// note: 7 stored wires end on pins the file does not list and are not shown
BCV_Loop.DeadBand := SEL(BCV_Loop.DeadBand = 0.0, BCV_Loop.DeadBand, 0.1);
BCV_Loop.Live_Target_EU := SEL(BCV_Loop.Mode=Temp_Loop_Modes.Step, BCV_Loop.Target_EU, SEL(HEATING, TT.EU-(BCV_Loop.DeadBand*1.5), TT.EU+(BCV_Loop.DeadBand*1.5)));
_w1 := (BCV_Loop.Mode = Temp_Loop_Modes.Crash) OR (BCV_Loop.Mode = Temp_Loop_Modes.Step);
_w2 := ABS(BCV_Loop.Target_EU - TT.EU);
ABS_Error := _w2;
(* _w2 * BCV_Loop.kp < 50; result not used *)
TON_2(IN := False OR _w2 < BCV_Loop.Window, PT := T#5s); // TON
_w3 := _w1 AND TON_2.Q;
In_Zone := _w3;
R_TRIG_0(CLK := _w1 AND _w3); // R_trig
IF R_TRIG_0.Q THEN _w4 := Temp_Loop_Modes.Auto; END_IF
BCV_Loop.Mode := _w4;
_w5 := REAL_TO_TIME(BCV_LOOP.Min_Cycle_S) * 1000;
_w6 := On_Seconds > BCV_LOOP.Min_Cycle_S;
_w7 := SEL(Heating, BCV_Loop.Live_Target_EU, BCV_Loop.Actual_EU);
_w8 := SEL(Heating, BCV_Loop.Actual_EU, BCV_Loop.Live_Target_EU);
TOF_0(IN := Permisive, PT := T#15s); // TOF
TON_3(IN := TOF_0.Q, PT := T#15s); // TON
_w9 := On_Seconds > BCV_LOOP.Max_Cycle_S - BCV_LOOP.Min_Cycle_S;
SR_0(SET1 := Loop_Disable, RESET := BCV_Loop.Mode=Temp_Loop_Modes.Idle); // SR
TP_1(IN := _w3, PT := T#5s); // TP
IF SR_0.Q1 THEN _w10 := Temp_Loop_Modes.Idle; END_IF
BCV_Loop.Mode := _w10;
_w11 := UINT_TO_TIME(BCV_Loop.Timer_Target_M) * 60000;
TOF_1(IN := (TT.Status.eStatus=eSensor_Status.Offline) OR (TT.Status.eStatus=eSensor_Status.Fault), PT := t#15s); // TOF
_w12 := (BCV_Loop.Mode=Temp_Loop_Modes.Auto_Paused) OR (BCV_Loop.Mode=Temp_Loop_Modes.Idle) OR NOT TON_3.Q OR SR_0.Q1 OR (BCV_Loop.Status=Temp_Loop_Status.Timer_Expired) OR TOF_1.Q;
_w13 := _w12 OR (_w12 OR TP_1.Q);
PID_Reset := _w13;
FT_PIDW_0(
    IN := SEL(_w12, _w8, _w7) - _w7,
    KP := BCV_Loop.kp,
    TN := BCV_Loop.TN,
    TV := BCV_Loop.TV,
    LIM_L := 0,
    LIM_H := 100,
    RST := _w13); // BURKERT_OSCAT_BASIC.FT_PIDW
BCV_Loop.Limiter := FT_PIDW_0.LIM;
_w14 := SEL(PID_Reset, SEL(BCV_Loop.Mode=Temp_Loop_Modes.Crash, FT_PIDW_0.Y, 100.0), 0.0);
BCV_Loop.Load_EU := _w14;
_w15 := _w14 * ((BCV_Loop.Max_Cycle_S/100.0));
On_Seconds := _w15;
GEN_PULSE_0(
    ENQ := _w6,
    PTH := REAL_TO_TIME(_w15) * 1000,
    PTL := REAL_TO_TIME(BCV_LOOP.Max_Cycle_S - _w15) * 1000); // BURKERT_OSCAT_BASIC.GEN_PULSE
_w16 := _w6 AND GEN_PULSE_0.Q;
TP_0(IN := _w16, PT := _w5); // TP
_w17 := (TP_0.Q OR _w16 OR _w9) AND NOT Loop_Disable AND NOT (BCV_Loop.Mode=Temp_Loop_Modes.Idle);
BCV_Loop.Output := _w17;
BCV.PLC_CMD := _w17;
_w18 := (BCV_Loop.Mode=Temp_Loop_Modes.Profile) AND (BCV_Loop.Timer_Target_M>0) AND NOT _w13 AND NOT Profile_Reset;
TON_0(IN := _w18, PT := _w11); // TON
Current_Minute := TIME_TO_UINT(TON_0.ET / 60000);
BCV_Loop.Timer_Remaining_s := TIME_TO_UINT((_w11 - TON_0.ET) / 1000);
TT.Alarm_Config.Setpoints.Hi_Hi_Alarm := SEL(NOT _w12, TT.Alarm_Config.Setpoints.Hi_Hi_Alarm, BCV_Loop.Live_Target_EU+(BCV_Loop.Window*2));
_w19 := (TT.Status.eStatus=eSensor_Status.Offline) OR (TT.Status.eStatus=eSensor_Status.Offline);
Loop_Disable := External_Fault OR (TT.Status.eStatus=eSensor_Status.FORCED) OR (BCV.Mode<>eBCV_Modes.Auto) OR _w19;
TT.Alarm_Config.Setpoints.Hi_Warn := SEL(NOT _w12, TT.Alarm_Config.Setpoints.Hi_Warn, BCV_Loop.Live_Target_EU+(BCV_Loop.Window));
TT.Alarm_Config.Setpoints.Low_warn := SEL(NOT _w12, TT.Alarm_Config.Setpoints.Low_warn, BCV_Loop.Live_Target_EU-(BCV_Loop.Window));
TT.Alarm_Config.Setpoints.Low_Low_Alarm := SEL(NOT _w12, TT.Alarm_Config.Setpoints.Low_Low_Alarm, BCV_Loop.Live_Target_EU-(BCV_Loop.Window*2));
BCV_Loop.Status := SEL(BCV.Mode<>eBCV_Modes.Auto, SEL(TT.Status.eStatus=eSensor_Status.FORCED, SEL(External_Fault, SEL(_w19, SEL(BCV_Loop.Mode=Temp_Loop_Modes.Auto_Paused, SEL(BCV_Loop.Mode=Temp_Loop_Modes.Idle, SEL(TT.Status.eStatus=eSensor_Status.Low_Low_Alarm, SEL(TT.Status.eStatus=eSensor_Status.Low_Warning, SEL(TT.Status.eStatus=eSensor_Status.HiHi_Alarm, SEL(TT.Status.eStatus=eSensor_Status.High_Warning, SEL(TON_0.Q, SEL(_w18, SEL(BCV_Loop.Mode=Temp_Loop_Modes.Auto, SEL(Permisive, Temp_Loop_Status.Pre_Start, Temp_Loop_Status.Ramping), Temp_Loop_Status.Auto), Temp_Loop_Status.Timed), Temp_Loop_Status.Timer_Expired), Temp_Loop_Status.HiHi_Warning), Temp_Loop_Status.HiHi_Alarm), Temp_Loop_Status.LoLo_Warning), Temp_Loop_Status.LoLo_Alarm), Temp_Loop_Status.Idle), Temp_Loop_Status.Paused), Temp_Loop_Status.Fault), Temp_Loop_Status.External_Fault), Temp_Loop_Status.Sensor_Forced), Temp_Loop_Status.Valve_Not_auto);
BCV_Loop.Actual_EU := TT.EU;
BCV_Loop.Error_EU := SEL(BCV_Loop.Mode=Temp_Loop_Modes.Idle, TT.EU - BCV_Loop.Target_EU, 0.0);
BCV_Loop.Int_Out := FT_PIDW_0.YI;
BCV_Loop.Diff_Out := FT_PIDW_0.diff.out;
TT.Alarm_Config.Silence := BCV_Loop.Mode=Temp_Loop_Modes.Idle;
R_TRIG_3(CLK := BCV_Loop.Mode=Temp_Loop_Modes.Profile); // R_trig
_w20 := R_TRIG_3.Q;
IF _w20 THEN _w21 := 0; END_IF
BCV_Loop.Temp_Profile.Index := _w21;
_w22 := (BCV_Loop.Mode=Temp_Loop_Modes.Profile) AND (BCV_Loop.Timer_Remaining_s=1) AND NOT (BCV_Loop.Temp_Profile.Index=4);
IF _w22 THEN _w23 := BCV_Loop.Temp_Profile.Index+1; END_IF
BCV_Loop.Temp_Profile.Index := _w23;
_w24 := (_w20 OR _w22) AND NOT (BCV_Loop.Temp_Profile.Time_m[BCV_Loop.Temp_Profile.Index]=0);
IF _w24 THEN _w25 := BCV_Loop.Temp_Profile.Time_m[BCV_Loop.Temp_Profile.Index]; END_IF
BCV_Loop.Timer_Target_M := _w25;
_w26 := _w24;
IF _w26 THEN _w27 := BCV_Loop.Temp_Profile.Target[BCV_Loop.Temp_Profile.Index]; END_IF
Profile_Reset := _w26;
BCV_Loop.Target_EU := _w27;
// TRUE: input not connected
// Temp_Loop_Status.Idle: input not connected

END_FUNCTION_BLOCK

// 20 Program Organization Units/FIT_DINT_UDBF
FUNCTION_BLOCK FIT_DINT_UDBF
VAR_INPUT
	Count:DINT;
	Frequency:REAL;
END_VAR

VAR_OUTPUT
	Reset:BOOL;
END_VAR

VAR
	R_Trig_0: R_Trig;
	COUNT_REAL: LREAL;
	Total:LREAL;
	FREQUENCY_REAL: REAL;
	Rate_Sec:REAL;
END_VAR
VAR_IN_OUT
	FIT:FIT_DUT;
END_VAR
VAR // added by the converter: edge detectors and wires of the graphical bodies
    _w1, _w2 : BOOL;
END_VAR

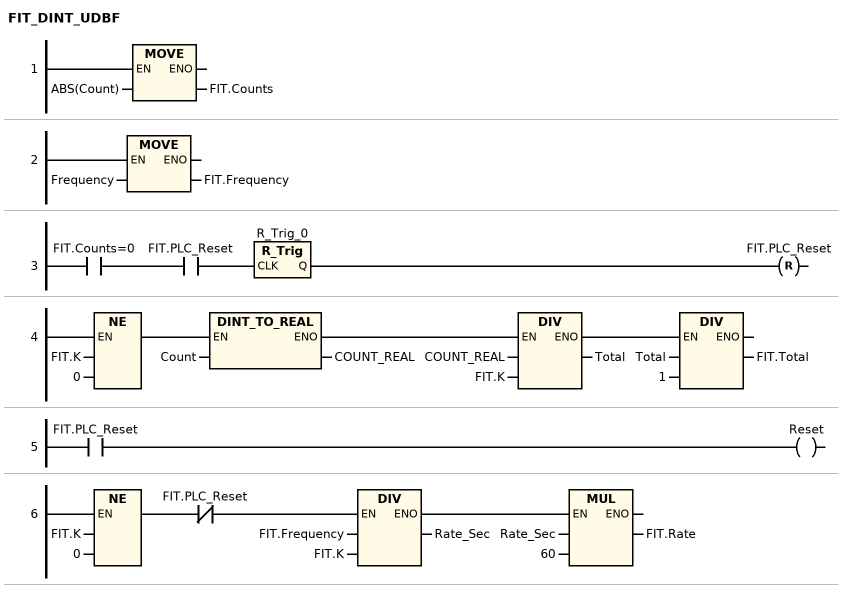
// NETWORK 1
FIT.Counts := ABS(Count);

// NETWORK 2
FIT.Frequency := Frequency;

// NETWORK 3
R_Trig_0(CLK := (FIT.Counts=0) AND FIT.PLC_Reset); // R_Trig
FIT.PLC_Reset R= R_Trig_0.Q;

// NETWORK 4
//   Total: K : REAL;
//   FIT.Total: K : REAL;
_w1 := FIT.K <> 0;
IF _w1 THEN COUNT_REAL := DINT_TO_REAL(Count); END_IF
IF _w1 THEN Total := COUNT_REAL / FIT.K; END_IF
IF _w1 THEN FIT.Total := Total / 1; END_IF

// NETWORK 5
Reset := FIT.PLC_Reset;

// NETWORK 6
_w2 := FIT.K <> 0 AND NOT FIT.PLC_Reset;
IF _w2 THEN Rate_Sec := FIT.Frequency / FIT.K; END_IF
IF _w2 THEN FIT.Rate := Rate_Sec * 60; END_IF

END_FUNCTION_BLOCK

// 20 Program Organization Units/FLOWave_UDFB
FUNCTION_BLOCK FLOWave_UDFB
VAR_INPUT
	//Reset_T1:BOOL;
	//Reset_T2:BOOL;
	//Can_Node:BYTE;
	RX:ARRAY[0..24] OF WORD;
	
	
END_VAR
VAR_OUTPUT
	//SDO_Data:cSDO_DUT;
	TX:ARRAY[0..3] OF WORD;
END_VAR
VAR_IN_OUT
	//Can_SDO_Pointer:INT;
	FloWave:cFLOWave_DUT;
END_VAR
VAR
	R_TRIG_0: R_Trig;
	R1_MSG_Pointer: BYTE;
	R2_MSG_Pointer: BYTE;
	SDO_Index:INT;
	SDO_MSG_Pointer:INT;
	SDO_RX:Bytes_2_Real;
	R_TRIG_1: R_trig;
	R_TRIG_2: R_Trig;
	F_TRIG_0: F_Trig;
	RX_Array:ARRAY[0..19] OF REAL;
	
	ALARM_2_0: BURKERT_OSCAT_BASIC.ALARM_2;
	ALARM_2_1: BURKERT_OSCAT_BASIC.ALARM_2;
	ALARM_2_3: BURKERT_OSCAT_BASIC.ALARM_2;
	tmp_Count1: REAL;
	tmp_Count2: REAL;
END_VAR

TX[3] := SEL(FloWave.FIT_2.PLC_Reset, 0, 256);
Alarms();
TX[1] := SEL(FloWave.M_Reset_2, 0, 256);
TX[0] := SEL(FloWave.M_Reset_1, 0, 256);
TX[2] := SEL(FloWave.FIT_1.PLC_Reset, 0, 256);
Translate();

ACTION Alarms:
ALARM_2_1(
    X := FloWave.Temp,
    LO_1 := floWave.Alarm_Config[1].Low_warn,
    HI_1 := floWave.Alarm_Config[1].Hi_Warn,
    LO_2 := floWave.Alarm_Config[1].Low_Low_Alarm,
    HI_2 := floWave.Alarm_Config[1].Hi_Hi_Alarm,
    HYS := 0.5); // BURKERT_OSCAT_BASIC.ALARM_2
ALARM_2_3(
    X := FloWave.Density_Factor,
    LO_1 := floWave.Alarm_Config[2].Low_warn,
    HI_1 := floWave.Alarm_Config[2].Hi_Warn,
    LO_2 := floWave.Alarm_Config[2].Low_Low_Alarm,
    HI_2 := floWave.Alarm_Config[2].Hi_Hi_Alarm,
    HYS := 0.5); // BURKERT_OSCAT_BASIC.ALARM_2
ALARM_2_0(
    X := FloWave.Concentration_2,
    LO_1 := floWave.Alarm_Config[0].Low_warn,
    HI_1 := floWave.Alarm_Config[0].Hi_Warn,
    LO_2 := floWave.Alarm_Config[0].Low_Low_Alarm,
    HI_2 := floWave.Alarm_Config[0].Hi_Hi_Alarm,
    HYS := 0.1); // BURKERT_OSCAT_BASIC.ALARM_2
ALARM_2_0(
    X := FloWave.Concentration_1,
    LO_1 := floWave.Alarm_Config[0].Low_warn,
    HI_1 := floWave.Alarm_Config[0].Hi_Warn,
    LO_2 := floWave.Alarm_Config[0].Low_Low_Alarm,
    HI_2 := floWave.Alarm_Config[0].Hi_Hi_Alarm,
    HYS := 0.1); // BURKERT_OSCAT_BASIC.ALARM_2
FloWave.Status := SEL(ALARM_2_0.Q2_HI OR ALARM_2_1.Q2_HI OR ALARM_2_3.Q2_HI OR ALARM_2_0.Q2_HI, SEL(ALARM_2_0.Q1_HI OR ALARM_2_1.Q1_HI OR ALARM_2_3.Q1_HI OR ALARM_2_0.Q1_HI, SEL(ALARM_2_0.Q2_LO OR ALARM_2_1.Q2_LO OR ALARM_2_3.Q2_LO OR ALARM_2_0.Q2_LO, SEL(ALARM_2_0.Q1_LO OR ALARM_2_1.Q1_LO OR ALARM_2_3.Q1_LO OR ALARM_2_0.Q1_LO, eFloWave_Status.OK, eFloWave_Status.Low_Warning), eFloWave_Status.Low_Low_Alarm), eFloWave_Status.High_Warning), eFloWave_Status.High_High_Alarm);
END_ACTION

ACTION Translate:
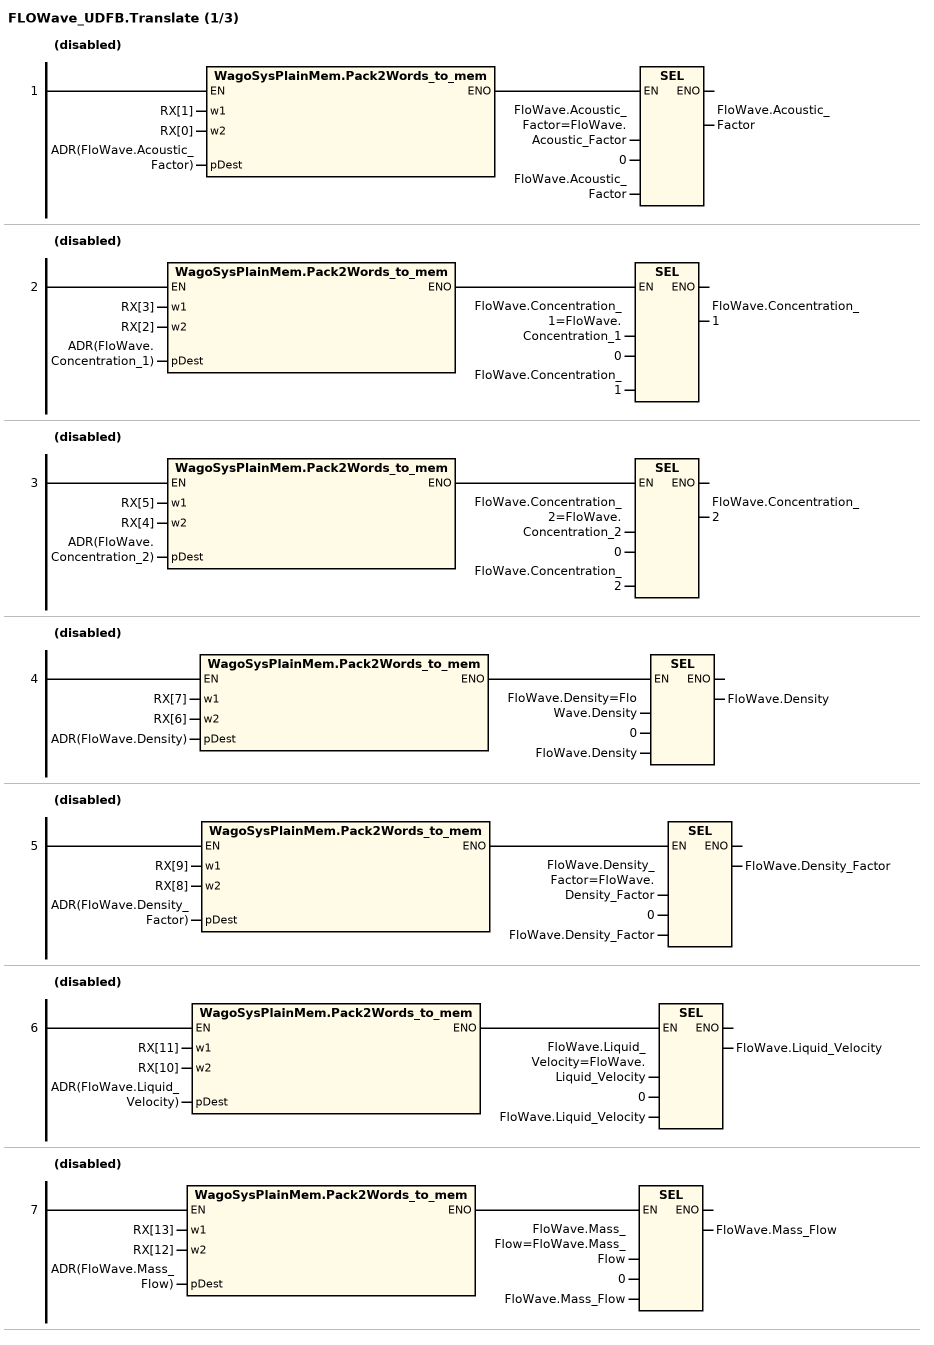
// NETWORK 1 (disabled)
// WagoSysPlainMem.Pack2Words_to_mem(w1 := RX[1], w2 := RX[0], pDest := ADR(FloWave.Acoustic_Factor));
// FloWave.Acoustic_Factor := SEL(FloWave.Acoustic_Factor=FloWave.Acoustic_Factor, 0, FloWave.Acoustic_Factor);

// NETWORK 2 (disabled)
// WagoSysPlainMem.Pack2Words_to_mem(w1 := RX[3], w2 := RX[2], pDest := ADR(FloWave.Concentration_1));
// FloWave.Concentration_1 := SEL(FloWave.Concentration_1=FloWave.Concentration_1, 0, FloWave.Concentration_1);

// NETWORK 3 (disabled)
// WagoSysPlainMem.Pack2Words_to_mem(w1 := RX[5], w2 := RX[4], pDest := ADR(FloWave.Concentration_2));
// FloWave.Concentration_2 := SEL(FloWave.Concentration_2=FloWave.Concentration_2, 0, FloWave.Concentration_2);

// NETWORK 4 (disabled)
// WagoSysPlainMem.Pack2Words_to_mem(w1 := RX[7], w2 := RX[6], pDest := ADR(FloWave.Density));
// FloWave.Density := SEL(FloWave.Density=FloWave.Density, 0, FloWave.Density);

// NETWORK 5 (disabled)
// WagoSysPlainMem.Pack2Words_to_mem(w1 := RX[9], w2 := RX[8], pDest := ADR(FloWave.Density_Factor));
// FloWave.Density_Factor := SEL(FloWave.Density_Factor=FloWave.Density_Factor, 0, FloWave.Density_Factor);

// NETWORK 6 (disabled)
// WagoSysPlainMem.Pack2Words_to_mem(w1 := RX[11], w2 := RX[10], pDest := ADR(FloWave.Liquid_Velocity));
// FloWave.Liquid_Velocity := SEL(FloWave.Liquid_Velocity=FloWave.Liquid_Velocity, 0, FloWave.Liquid_Velocity);

// NETWORK 7 (disabled)
// WagoSysPlainMem.Pack2Words_to_mem(w1 := RX[13], w2 := RX[12], pDest := ADR(FloWave.Mass_Flow));
// FloWave.Mass_Flow := SEL(FloWave.Mass_Flow=FloWave.Mass_Flow, 0, FloWave.Mass_Flow);

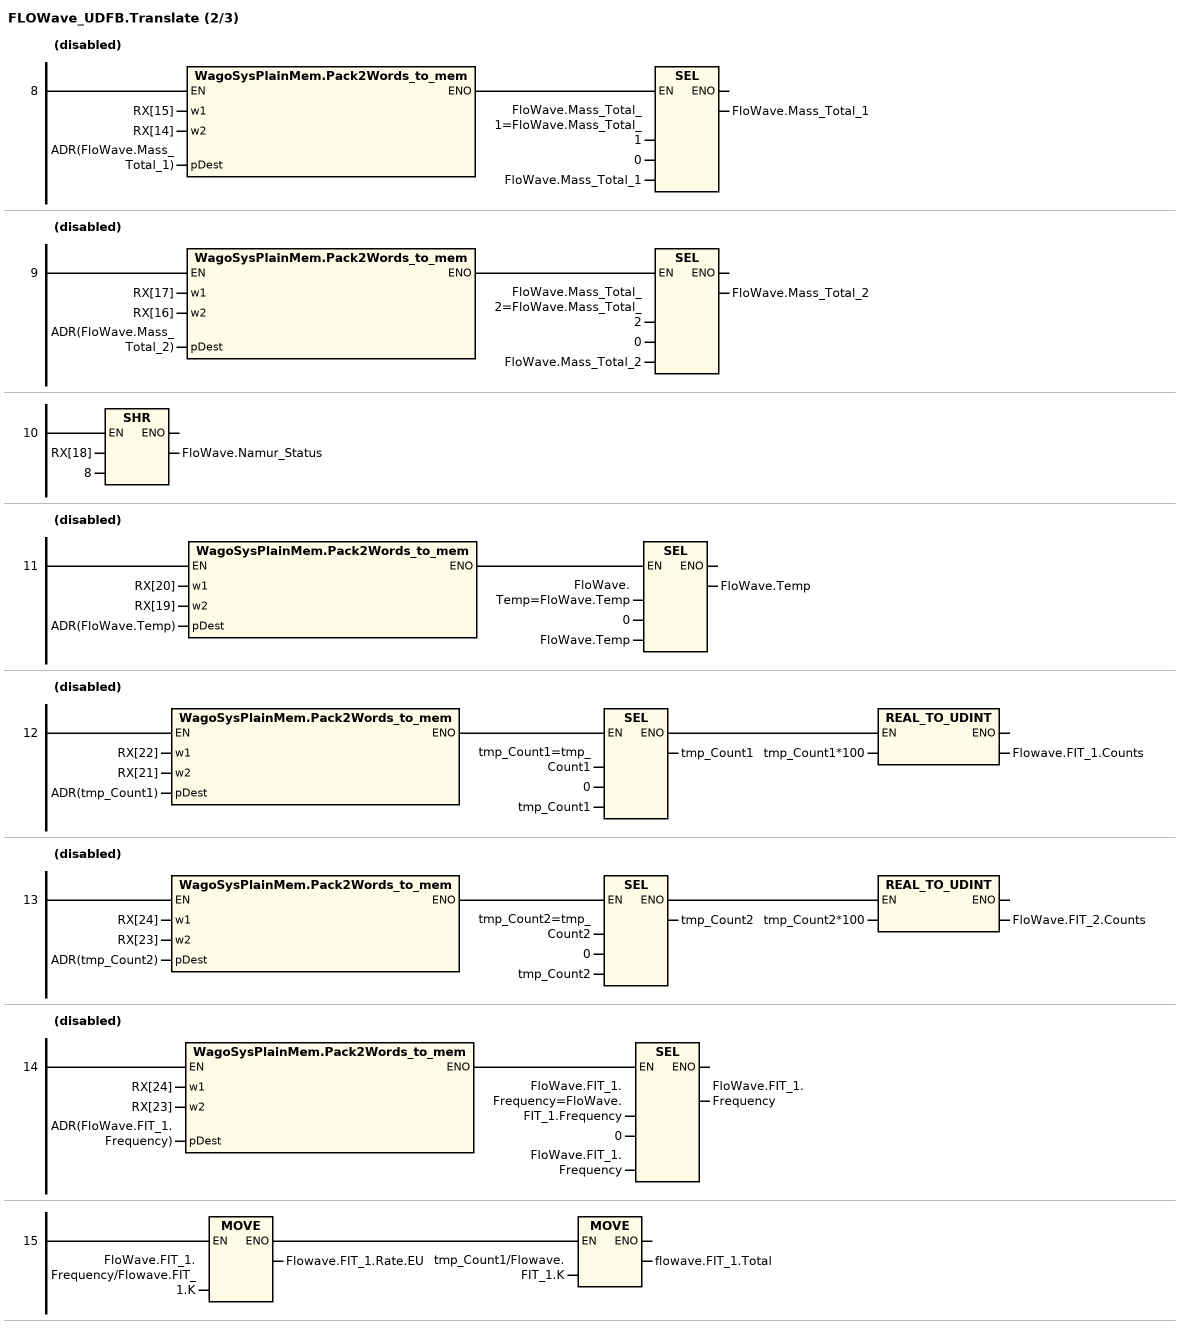
// NETWORK 8 (disabled)
// WagoSysPlainMem.Pack2Words_to_mem(w1 := RX[15], w2 := RX[14], pDest := ADR(FloWave.Mass_Total_1));
// FloWave.Mass_Total_1 := SEL(FloWave.Mass_Total_1=FloWave.Mass_Total_1, 0, FloWave.Mass_Total_1);

// NETWORK 9 (disabled)
// WagoSysPlainMem.Pack2Words_to_mem(w1 := RX[17], w2 := RX[16], pDest := ADR(FloWave.Mass_Total_2));
// FloWave.Mass_Total_2 := SEL(FloWave.Mass_Total_2=FloWave.Mass_Total_2, 0, FloWave.Mass_Total_2);

// NETWORK 10
FloWave.Namur_Status := SHR(RX[18], 8);

// NETWORK 11 (disabled)
// WagoSysPlainMem.Pack2Words_to_mem(w1 := RX[20], w2 := RX[19], pDest := ADR(FloWave.Temp));
// FloWave.Temp := SEL(FloWave.Temp=FloWave.Temp, 0, FloWave.Temp);

// NETWORK 12 (disabled)
// WagoSysPlainMem.Pack2Words_to_mem(w1 := RX[22], w2 := RX[21], pDest := ADR(tmp_Count1));
// tmp_Count1 := SEL(tmp_Count1=tmp_Count1, 0, tmp_Count1);
// Flowave.FIT_1.Counts := REAL_TO_UDINT(tmp_Count1*100);

// NETWORK 13 (disabled)
// WagoSysPlainMem.Pack2Words_to_mem(w1 := RX[24], w2 := RX[23], pDest := ADR(tmp_Count2));
// tmp_Count2 := SEL(tmp_Count2=tmp_Count2, 0, tmp_Count2);
// FloWave.FIT_2.Counts := REAL_TO_UDINT(tmp_Count2*100);

// NETWORK 14 (disabled)
// WagoSysPlainMem.Pack2Words_to_mem(w1 := RX[24], w2 := RX[23], pDest := ADR(FloWave.FIT_1.Frequency));
// FloWave.FIT_1.Frequency := SEL(FloWave.FIT_1.Frequency=FloWave.FIT_1.Frequency, 0, FloWave.FIT_1.Frequency);

// NETWORK 15
Flowave.FIT_1.Rate.EU := FloWave.FIT_1.Frequency/Flowave.FIT_1.K;
flowave.FIT_1.Total := tmp_Count1/Flowave.FIT_1.K;

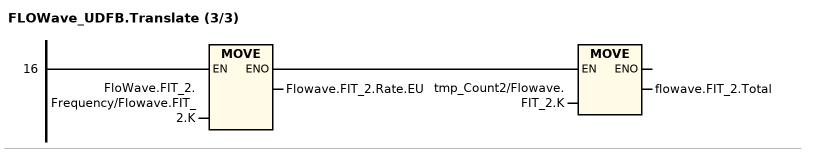
// NETWORK 16
Flowave.FIT_2.Rate.EU := FloWave.FIT_2.Frequency/Flowave.FIT_2.K;
flowave.FIT_2.Total := tmp_Count2/Flowave.FIT_2.K;
END_ACTION

END_FUNCTION_BLOCK

// 20 Program Organization Units/Tempered_Mix_eDip_UDFB
FUNCTION_BLOCK Tempered_Mix_eDip_UDFB
VAR_INPUT
	//Loop_ID:INT;
END_VAR
VAR_IN_OUT
	HW_ACV:eDip_8694_DUT;
	CW_ACV:eDip_8694_DUT;
	Temperature:AIT_DUT;
	FIT:FIT_DUT;
	Control:Mix_DUT;
END_VAR
VAR_OUTPUT
END_VAR
VAR
	R_TRIG_0: R_Trig;
	RATE_PID: BURKERT_OSCAT_BASIC.CTRL_PID;
	
	Temp_PID: BURKERT_OSCAT_BASIC.CTRL_PID;
	TON_0: TON;
	Stage_Delay: TIME := T#2s;
	TON_1: TON;
	TON_2: TON;
	SRAMP_0: BURKERT_OSCAT_BASIC.SRAMP;
	TON_3: TON;
	TON_4: TON;
	Ramp_Active: BOOL;
	Ramp_Target: REAL;
	TON_5: TON;
	TON_6: TON;
	R_TRIG_1: R_trig;
	Ramp_Start_Volume: REAL;
	Ramp_Volume: REAL;
	R_TRIG_2: R_Trig;
	R_TRIG_3: R_Trig;
	PID_0: Util.PID;
	R_TRIG_4: R_Trig;
	R_TRIG_5:R_trig;
	Live_Rate:Real;
	
END_VAR
VAR // added by the converter: edge detectors and wires of the graphical bodies
    _w1, _w2, _w3, _w4, _w5, _w6, _w11, _w13, _w14, _w15, _w16, _w17, _w19, _w20, _w23, _w25, _w27, _w33, _w34, _w35, _w37 : ANY;
    _w7, _w8, _w9, _w10, _w12, _w18, _w21, _w22, _w24, _w26, _w28, _w30, _w31, _w32, _w36, _w38 : BOOL;
    _w29 : REAL;
END_VAR

// note: 17 stored wires end on pins the file does not list and are not shown
IF NOT (HW_ACV.Mode=ACv_Modes.Auto) THEN _w1 := Mix_Status.HW_Valve_Not_Ready; END_IF
Control.Status := _w1;
IF NOT (CW_ACV.Mode=ACv_Modes.Auto) THEN _w2 := Mix_Status.CW_Valve_Not_Ready; END_IF
Control.Status := _w2;
Control.Actual_Rate_EU := FIT.Rate;
_w3 := (Control.Mode=Mix_Modes.IDlE) OR (Control.STATUS>Mix_Status.Batch_Ending) OR (Control.Mode=Mix_Modes.Pause);
RATE_PID(
    ACT := FIT.Rate,
    SET := Live_Rate,
    SUP := 0.1,
    OFS := 0.0,
    M_I := 0.0,
    MAN := _w3,
    RST := _w3,
    KP := Control.Config.Flow_KP,
    TN := Control.Config.Flow_TN,
    TV := Control.Config.Flow_TV,
    LL := 0,
    LH := 100.0); // BURKERT_OSCAT_BASIC.CTRL_PID
Control.Flow_CV := RATE_PID.Y;
R_TRIG_2(CLK := _w3 AND (Temperature.Mode.eMode<>AIT_Modes.Forced)); // R_Trig
IF R_TRIG_2.Q THEN _w4 := AIT_Modes.Alarms_Disabled; END_IF
Temperature.Mode.eMode := _w4;
Control.Actual_Temp_EU := Temperature.EU;
_w5 := (Control.Mode=Mix_Modes.IDlE) OR (Control.Mode=Mix_Modes.Rate_Only) OR (Control.STATUS>Mix_Status.Batch_Ending) OR (Control.STATUS=Mix_Status.Start_Flow) OR (Control.STATUS=Mix_Status.Fit_Reset) OR (Control.Mode=Mix_Modes.Pause);
PID_0(
    ACTUAL := Temperature.EU,
    SET_POINT := Control.Config.TARGET_C,
    KP := Control.Config.Temp_KP,
    TN := Control.Config.Temp_TN,
    TV := Control.Config.Temp_TV,
    Y_MANUAL := 0,
    Y_OFFSET := 0,
    Y_MIN := -100,
    Y_MAX := 100,
    MANUAL := _w5,
    RESET := _w5); // Util.PID
Control.Temp_CV := SEl(Control.Mode=Mix_Modes.Cold_Only, SEl(Control.Mode=Mix_Modes.Hot_Only, PID_0.Y, 100), -100);
SRAMP_0(
    X := Ramp_Target,
    A_UP := Control.Config.Ramp_Rate,
    A_DN := 0-Control.config.Ramp_Rate,
    VU_MAX := Control.config.Max_Flow,
    VD_MAX := 0-Control.config.Max_Flow,
    LIMIT_HIGH := Control.config.Max_Flow,
    LIMIT_LOW := Control.Config.Min_Flow,
    RST := Control.Mode=Mix_Modes.IDlE); // BURKERT_OSCAT_BASIC.SRAMP
Live_Rate := SRAMP_0.Y;
IF Control.Mode=Mix_Modes.IDlE THEN _w6 := Mix_Status.IDle; END_IF
Control.STATUS := _w6;
R_TRIG_0(CLK := (Control.Mode=Mix_Modes.Auto) OR (Control.Mode=Mix_Modes.Hot_Only) OR (Control.Mode=Mix_Modes.Cold_Only) OR (Control.Mode=Mix_Modes.Quick_Start)); // R_Trig
Control.STATUS := SEL(R_TRIG_0.Q, Control.STATUS, Mix_Status.Fit_Reset);
Control.Actual_Volume_EU := FIT.Total;
_w7 := Control.STATUS = Mix_Status.Fit_Reset;
IF _w7 THEN _w8 := False; END_IF
Ramp_active := _w8;
_w9 := NOT (FIT.Total>0.1) AND _w7;
FIT.PLC_Reset := SEL(_w7 AND (FIT.Total>0.1), SEL(_w9, FIT.PLC_Reset, False), True);
_w10 := _w9;
IF _w10 THEN _w11 := Mix_Status.Start_Flow; END_IF
_w12 := _w10;
IF _w12 THEN _w13 := SEL(Control.Mode=Mix_Modes.Hot_Only, _w11, Mix_Status.Temperature_OK); END_IF
IF _w12 THEN _w14 := SEL(Control.Mode=Mix_Modes.Hot_Only, _w13, Mix_Status.Temperature_OK); END_IF
Control.STATUS := _w14;
_w15 := Control.Temp_CV / 100.0;
_w16 := LIMIT(0, Control.Flow_CV * (1.0 + _w15), 100);
Control.HW_CMD := _w16;
HW_ACV.PLC_CMD := _w16;
_w17 := LIMIT(0, Control.Flow_CV * (1.0 - _w15), 100);
Control.CW_CMD := _w17;
CW_ACV.PLC_CMD := _w17;
_w18 := Control.STATUS = Mix_Status.Start_Flow;
IF _w18 THEN _w19 := Control.Config.Min_Flow; END_IF
Ramp_Target := _w19;
TON_0(IN := _w18 AND (Control.Actual_Rate_EU > (Control.Config.Min_Flow*0.8) OR (Control.Mode=Mix_Modes.Quick_Start)), PT := Stage_Delay); // TON
Control.STATUS := SEL(TON_0.Q, Control.STATUS, Mix_Status.Flow_Detected);
TON_1(IN := Control.STATUS = Mix_Status.Flow_Detected, PT := Stage_Delay); // TON
R_TRIG_3(CLK := (Temperature.Mode.eMode<>AIT_Modes.Forced) AND TON_1.Q); // R_Trig
IF R_TRIG_3.Q THEN _w20 := TT_Modes.Active; END_IF
Temperature.Mode.eMode := _w20;
Control.STATUS := SEL(TON_1.Q, Control.STATUS, Mix_Status.Start_temperature);
Temperature.Alarm_Config.Setpoints.Hi_Hi_Alarm := Control.Config.TARGET_C+(Control.Config.TEMP_WINDOW*4);
Temperature.Alarm_Config.Setpoints.Hi_Warn := Control.Config.TARGET_C+(Control.Config.TEMP_WINDOW*2);
Temperature.Alarm_Config.Setpoints.Low_warn := Control.Config.TARGET_C-(Control.Config.TEMP_WINDOW*2);
Temperature.Alarm_Config.Setpoints.Low_Low_Alarm := Control.Config.TARGET_C-(Control.Config.TEMP_WINDOW*4);
TON_2(IN := Control.STATUS = Mix_Status.Start_temperature AND (Control.Actual_Temp_EU > (Control.Config.TARGET_C-Control.Config.TEMP_WINDOW) OR (Control.Mode=Mix_Modes.Quick_Start)), PT := Stage_Delay); // TON
Control.STATUS := SEL(TON_2.Q, Control.STATUS, Mix_Status.Temperature_OK);
TON_3(IN := Control.STATUS = Mix_Status.Temperature_OK, PT := Stage_Delay); // TON
Control.STATUS := SEL(TON_3.Q, Control.STATUS, Mix_Status.Foundation_Rate);
_w21 := Control.STATUS = Mix_Status.Foundation_Rate;
Ramp_Active := SEL(_w21, Ramp_Active, True);
_w22 := _w21;
IF _w22 THEN _w23 := Control.Config.Foundation_Rate; END_IF
Ramp_Target := _w23;
Control.STATUS := SEL(_w22 AND (Control.Actual_Rate_EU >= (Control.Config.Foundation_Rate*0.9) OR (Control.Mode=Mix_Modes.Quick_Start)), Control.STATUS, Mix_Status.Foundation_Rate_OK);
TON_4(IN := Control.STATUS = Mix_Status.Foundation_Rate_OK AND (FIT.Total >= Control.Config.Foundation_Volume OR (Control.Mode=Mix_Modes.Quick_Start)), PT := Stage_Delay); // TON
Control.STATUS := SEL(TON_4.Q, Control.STATUS, Mix_Status.Foundation_Amount_Complete);
R_TRIG_5(CLK := Control.Mode=Mix_Modes.Resume); // R_trig
TON_5(IN := Control.STATUS = Mix_Status.Foundation_Amount_Complete, PT := Stage_Delay); // TON
Control.STATUS := SEL(R_TRIG_5.Q OR TON_5.Q, Control.STATUS, Mix_Status.Main_Rate);
_w24 := Control.STATUS = Mix_Status.Main_Rate;
R_TRIG_1(CLK := _w24); // R_trig
IF R_TRIG_1.Q THEN _w25 := Control.Actual_Volume_EU; END_IF
Ramp_Start_Volume := _w25;
_w26 := _w24;
IF _w26 THEN _w27 := Control.Config.TARGET_lpm; END_IF
Ramp_Target := _w27;
_w28 := _w26 AND Control.Actual_Rate_EU >= (Control.Config.TARGET_lpm*0.9);
Control.STATUS := SEL(_w28, Control.STATUS, Mix_Status.Main_Rate_OK);
IF _w28 THEN _w29 := Control.Actual_Volume_EU - Ramp_Start_Volume; END_IF
Ramp_Volume := _w29;
_w30 := Control.STATUS = Mix_Status.Main_Rate_OK;
TON_6(IN := _w30, PT := Stage_Delay); // TON
Control.STATUS := SEL(TON_6.Q, Control.STATUS, Mix_Status.Grain_Dispense);
_w31 := Control.STATUS = Mix_Status.Grain_Dispense;
_w32 := _w31;
IF _w32 THEN _w33 := Control.Config.TARGET_C; END_IF
Control.Config.TARGET_C := _w33;
IF _w32 THEN _w34 := Control.Config.TARGET_lpm; END_IF
Ramp_Target := _w34;
Control.STATUS := SEL(_w31 AND Control.Actual_Volume_EU >= (Control.Config.TARGET_L-Control.Config.Foundation_Volume), Control.STATUS, Mix_Status.Batch_Ending);
IF Control.Actual_Rate_EU>0.5 THEN _w35 := ((Control.Config.TARGET_L-Control.Config.Foundation_Volume) - Control.Actual_Volume_EU) / (Control.Actual_Rate_EU/60); END_IF
Control.Grain_ETA_S := REAL_TO_INT(_w35);
_w36 := Control.STATUS = Mix_Status.Batch_Ending;
IF _w36 THEN _w37 := Control.Config.Foundation_Rate; END_IF
Ramp_Target := _w37;
_w38 := (_w24 OR _w30 OR _w31 OR _w36) AND Control.Actual_Volume_EU >= Control.Config.TARGET_L;
Ramp_Active := SEl(_w38, Ramp_Active, FALSE);
Control.STATUS := SEL(_w38, Control.STATUS, Mix_Status.Batch_Complete);
// 0.1: input not connected

END_FUNCTION_BLOCK

// 20 Program Organization Units/Transfer_ACV_FIT_UDFB
FUNCTION_BLOCK Transfer_ACV_FIT_UDFB
VAR_INPUT
	//Index:INT;
	LOCK_OUT:BOOL:=FALSE;
	
END_VAR
VAR_OUTPUT
END_VAR
VAR
	Paused:BOOL;
	Idle_return:BOOL;
	Transfer_Running:BOOL;
	Complete:BOOL;
	ACV_Not_Ready:BOOL;
	//VFD_Not_Ready:BOOL;
	BCV_Not_Ready:BOOL;
	Time_Complete:BOOL;
	FIT_Reset_Complete:BOOL;
	//Pump_Start:BOOL;
	Lockout_Active:BOOL;
	Error:BOOL;
	//Flow_Mode:BOOL;
	Batch_Complete:BOOL;
	//Enable_pump:BOOL;
	
	PID_CV:REAL;
	
	
	
	
	SR2: SR;
	TON_0: TON;
	CTRL_PID_1: BURKERT_OSCAT_BASIC.CTRL_PID;
	R_TRIG_0: R_trig;
	TON_10: TON;
	SR_10: SR;
	RS_11: RS;
	TON_12: TON;
	F_TRIG_10: F_Trig;
	TP11: TP;
END_VAR

VAR_IN_OUT
	Transfer:FIT_VFD_Transfer_DUT;
	//VFD:VFD_Vacon_DUT;
	ACV:ACV_DUT;
	FIT:FIT_DUT;
	
END_VAR
VAR // added by the converter: edge detectors and wires of the graphical bodies
    _w1, _w2, _w6, _w17, _w19 : ANY;
    _w3, _w4, _w5, _w7, _w8, _w9, _w10, _w11, _w12, _w13, _w14, _w15, _w16, _w18, _w20 : BOOL;
END_VAR

